TYPE S_Panel_Hardware :
STRUCT
	(* Botones y alarmas específicos de una estación *)
 
	PE_Seta					AT %I*: BOOL;
	POC_PulsadorReset		AT %I*: BOOL; // POC Botón azul está pulsado (PO Conectada)
	PM_PulsadorMarcha		AT %I*: BOOL; // PM - Pulsador de marcha (verde)
	LM_LamparaMarcha		AT %Q*: BOOL; // LM - Lámpara marcha (verde)
	PS_PulsadorStop			AT %I*: BOOL; // PS - Pulsador de parada (rojo)
	LS_LamparaStop			AT %Q*: BOOL; // DUDAS - LA - Lámpara de alarma o lámpara de stop
	SM_SelecAutoManual	 	AT %I*: BOOL; // SM - Selector modo auto/man
	//ResetBoton				: BOOL; // DUDAS - HAY QUE VINCULARLO?
	//ResetLuzAzul			AT %Q*: BOOL; // DUDAS - HAY QUE VINCULARLO?

	AS_AvisadorSonoro		AT %Q*: BOOL; // AS - Avisador Sonoro
	LA_LamparaAlarma		AT %Q*: BOOL; // DUDAS - Es lo mismo que falta de material?
	DPO_DesconectaPO		AT %Q*: BOOL; // DPO - Desconecta PO
END_STRUCT
END_TYPE

(* stored: Version 1.1.0.1, ProductVersion 3.1.4024.6
   DUT S_Panel_Hardware: Id {30d6b7af-3833-46ea-8124-23bb4386cc10} *)
